INTERFACE I_Interface

PROPERTY SomeProperty : INT
GET
END_GET
SET
END_SET
END_PROPERTY

END_INTERFACE

(* stored: Version 1.1.0.1, ProductVersion 3.1.4024.10
   Itf I_Interface: Id {203124bb-05dd-41ab-8d91-438e10f5a30d}
   Property SomeProperty: Id {f9d73e21-fe2f-4fd4-9678-962e0d3e4644}
   Get Get: Id {114e75f4-8ba8-44d7-a8cf-2a2d45238614}
   Set Set: Id {9db3a523-8f24-4eb7-b184-675dc73ee74a} *)
